SPLINE
SPL {X  -141.803, Y  +311.593, Z    +0.000, E1   +37.608, E3 +232094.448}
SPL {X  -154.548, Y  +344.290, Z    +0.000, E1   +25.264, E3 +232118.932}
SPL {X  -159.249, Y  +370.212, Z    +0.000, E1   +11.801, E3 +232126.964}
SPL {X  -159.987, Y  +383.623, Z    +0.000, E1    +3.169, E3 +232128.717}
SPL {X  -160.000, Y  +388.238, Z    +0.000, E1    -0.420, E3 +232128.928}
SPL {X  -160.000, Y  +392.418, Z    +0.000, E1    -5.131, E3 +232129.169}
SPL {X  -160.000, Y  +399.157, Z    +0.000, E1   -14.351, E3 +232129.985}
SPL {X  -160.000, Y  +411.277, Z    +0.000, E1   -30.487, E3 +232132.763}
SPL {X  -160.000, Y  +452.990, Z    +0.000, E1   -53.470, E3 +232154.127}
SPL {X  -160.000, Y  +539.177, Z    +0.000, E1   -59.280, E3 +232232.454}
SPL {X  -160.000, Y  +554.731, Z    +0.000, E1   -59.281, E3 +232252.098}
SPL {X  -160.000, Y  +572.172, Z    +0.000, E1   -59.312, E3 +232274.061}
SPL {X  -160.000, Y  +589.502, Z    +0.000, E1   -59.284, E3 +232295.999}
SPL {X  -160.000, Y  +604.577, Z    +0.000, E1   -59.272, E3 +232315.058}
SPL {X  -160.000, Y  +620.386, Z    +0.000, E1   -59.294, E3 +232334.986}
SPL {X  -160.000, Y  +636.664, Z    +0.000, E1   -59.282, E3 +232355.575}
SPL {X  -160.000, Y  +654.257, Z    +0.000, E1   -59.312, E3 +232377.754}
SPL {X  -160.000, Y  +671.385, Z    +0.000, E1   -59.278, E3 +232399.443}
SPL {X  -159.497, Y  +687.081, Z    +0.000, E1   -59.218, E3 +232419.770}
SPL {X  -157.563, Y  +702.220, Z    +0.000, E1   -58.916, E3 +232440.931}
SPL {X  -154.922, Y  +714.390, Z    +0.000, E1   -58.446, E3 +232459.125}
SPL {X  -151.559, Y  +725.681, Z    +0.000, E1   -57.922, E3 +232476.756}
SPL {X  -147.777, Y  +735.736, Z    +0.000, E1   -57.226, E3 +232493.250}
SPL {X  -143.698, Y  +744.763, Z    +0.000, E1   -56.526, E3 +232508.527}
SPL {X  -138.992, Y  +753.654, Z    +0.000, E1   -55.630, E3 +232524.104}
SPL {X  -122.847, Y  +776.912, Z    +0.000, E1   -47.251, E3 +232633.787}
ENDSPLINE

SPLINE
SPL {X  -149.319, Y  +731.879, Z    +0.000, E1   -32.249, E3 +232728.173}
SPL {X  -158.304, Y  +697.637, Z    +0.000, E1   -16.440, E3 +232742.824}
SPL {X  -159.863, Y  +681.030, Z    +0.000, E1    -6.312, E3 +232745.766}
SPL {X  -160.000, Y  +673.530, Z    +0.000, E1    -1.059, E3 +232746.273}
SPL {X  -160.000, Y  +670.245, Z    +0.000, E1    +2.042, E3 +232746.386}
SPL {X  -160.000, Y  +663.790, Z    +0.000, E1   +10.467, E3 +232746.911}
SPL {X  -160.000, Y  +655.457, Z    +0.000, E1   +22.866, E3 +232748.273}
SPL {X  -160.000, Y  +644.540, Z    +0.000, E1   +36.054, E3 +232751.304}
SPL {X  -160.000, Y  +601.495, Z    +0.000, E1   +56.174, E3 +232772.233}
SPL {X  -160.000, Y  +515.545, Z    +0.000, E1   +60.629, E3 +232847.627}
SPL {X  -160.000, Y  +503.330, Z    +0.000, E1   +60.630, E3 +232862.233}
SPL {X  -160.000, Y  +487.139, Z    +0.000, E1   +60.676, E3 +232881.501}
SPL {X  -160.000, Y  +466.770, Z    +0.000, E1   +60.698, E3 +232905.797}
SPL {X  -160.000, Y  +454.269, Z    +0.000, E1   +59.898, E3 +232926.048}
ENDSPLINE

SPLINE
SPL {X  -160.000, Y  +458.973, Z    +0.000, E1   +55.880, E3 +232946.966}
ENDSPLINE

SPLINE
SPL {X  -160.000, Y  +435.816, Z    +0.000, E1   +57.237, E3 +232970.642}
SPL {X  -160.000, Y  +411.824, Z    +0.000, E1   +58.675, E3 +232993.135}
SPL {X  -160.000, Y  +390.940, Z    +0.000, E1   +59.356, E3 +233015.163}
SPL {X  -159.620, Y  +374.678, Z    +0.000, E1   +59.299, E3 +233036.047}
SPL {X  -157.749, Y  +358.956, Z    +0.000, E1   +59.037, E3 +233057.745}
SPL {X  -154.809, Y  +345.275, Z    +0.000, E1   +58.527, E3 +233078.068}
SPL {X  -151.181, Y  +333.313, Z    +0.000, E1   +57.939, E3 +233096.777}
SPL {X  -146.730, Y  +321.901, Z    +0.000, E1   +57.169, E3 +233115.522}
SPL {X  -142.568, Y  +313.075, Z    +0.000, E1   +56.366, E3 +233130.644}
SPL {X  -139.172, Y  +306.763, Z    +0.000, E1   +55.717, E3 +233141.699}
SPL {X  -137.037, Y  +303.112, Z    +0.000, E1   +55.261, E3 +233148.245}
SPL {X  -123.439, Y  +283.902, Z    +0.000, E1   +48.158, E3 +233234.596}
ENDSPLINE

SPLINE
SPL {X  -141.803, Y  +311.593, Z    +0.000, E1   +37.608, E3 +233325.216}
SPL {X  -154.548, Y  +344.290, Z    +0.000, E1   +25.264, E3 +233349.699}
SPL {X  -159.249, Y  +370.212, Z    +0.000, E1   +11.801, E3 +233357.731}
SPL {X  -159.987, Y  +383.623, Z    +0.000, E1    +3.169, E3 +233359.484}
SPL {X  -160.000, Y  +388.238, Z    +0.000, E1    -0.420, E3 +233359.696}
SPL {X  -160.000, Y  +392.418, Z    +0.000, E1    -5.131, E3 +233359.936}
SPL {X  -160.000, Y  +399.157, Z    +0.000, E1   -14.351, E3 +233360.752}
SPL {X  -160.000, Y  +411.277, Z    +0.000, E1   -30.487, E3 +233363.530}
SPL {X  -160.000, Y  +452.990, Z    +0.000, E1   -53.470, E3 +233384.894}
SPL {X  -160.000, Y  +539.177, Z    +0.000, E1   -59.280, E3 +233463.221}
SPL {X  -160.000, Y  +554.731, Z    +0.000, E1   -59.281, E3 +233482.865}
SPL {X  -160.000, Y  +572.172, Z    +0.000, E1   -59.312, E3 +233504.828}
SPL {X  -160.000, Y  +589.502, Z    +0.000, E1   -59.284, E3 +233526.766}
SPL {X  -160.000, Y  +604.577, Z    +0.000, E1   -59.272, E3 +233545.826}
SPL {X  -160.000, Y  +620.386, Z    +0.000, E1   -59.294, E3 +233565.753}
SPL {X  -160.000, Y  +636.664, Z    +0.000, E1   -59.282, E3 +233586.343}
SPL {X  -160.000, Y  +654.257, Z    +0.000, E1   -59.312, E3 +233608.521}
SPL {X  -160.000, Y  +671.385, Z    +0.000, E1   -59.278, E3 +233630.210}
SPL {X  -159.497, Y  +687.081, Z    +0.000, E1   -59.218, E3 +233650.537}
SPL {X  -157.563, Y  +702.220, Z    +0.000, E1   -58.916, E3 +233671.699}
SPL {X  -154.922, Y  +714.390, Z    +0.000, E1   -58.446, E3 +233689.892}
SPL {X  -151.559, Y  +725.681, Z    +0.000, E1   -57.922, E3 +233707.523}
SPL {X  -147.777, Y  +735.736, Z    +0.000, E1   -57.226, E3 +233724.017}
SPL {X  -143.698, Y  +744.763, Z    +0.000, E1   -56.526, E3 +233739.294}
SPL {X  -138.992, Y  +753.654, Z    +0.000, E1   -55.630, E3 +233754.871}
SPL {X  -122.847, Y  +776.912, Z    +0.000, E1   -47.251, E3 +233864.554}
ENDSPLINE

SPLINE
SPL {X  -149.319, Y  +731.879, Z    +0.000, E1   -32.249, E3 +233958.941}
SPL {X  -158.304, Y  +697.637, Z    +0.000, E1   -16.440, E3 +233973.591}
SPL {X  -159.863, Y  +681.030, Z    +0.000, E1    -6.312, E3 +233976.533}
SPL {X  -160.000, Y  +673.530, Z    +0.000, E1    -1.059, E3 +233977.040}
SPL {X  -160.000, Y  +670.245, Z    +0.000, E1    +2.042, E3 +233977.153}
SPL {X  -160.000, Y  +663.790, Z    +0.000, E1   +10.467, E3 +233977.678}
SPL {X  -160.000, Y  +655.457, Z    +0.000, E1   +22.866, E3 +233979.040}
SPL {X  -160.000, Y  +644.540, Z    +0.000, E1   +36.054, E3 +233982.071}
SPL {X  -160.000, Y  +601.495, Z    +0.000, E1   +56.174, E3 +234003.000}
SPL {X  -160.000, Y  +515.545, Z    +0.000, E1   +60.629, E3 +234078.394}
SPL {X  -160.000, Y  +503.330, Z    +0.000, E1   +60.630, E3 +234093.000}
SPL {X  -160.000, Y  +487.139, Z    +0.000, E1   +60.676, E3 +234112.268}
SPL {X  -160.000, Y  +466.770, Z    +0.000, E1   +60.698, E3 +234136.564}
SPL {X  -160.000, Y  +454.269, Z    +0.000, E1   +59.898, E3 +234156.815}
ENDSPLINE

SPLINE
SPL {X  -160.000, Y  +458.973, Z    +0.000, E1   +55.880, E3 +234177.733}
ENDSPLINE

SPLINE
SPL {X  -160.000, Y  +435.816, Z    +0.000, E1   +57.237, E3 +234201.409}
SPL {X  -160.000, Y  +411.824, Z    +0.000, E1   +58.675, E3 +234223.903}
SPL {X  -160.000, Y  +390.940, Z    +0.000, E1   +59.356, E3 +234245.930}
SPL {X  -159.620, Y  +374.678, Z    +0.000, E1   +59.299, E3 +234266.814}
SPL {X  -157.749, Y  +358.956, Z    +0.000, E1   +59.037, E3 +234288.512}
SPL {X  -154.809, Y  +345.275, Z    +0.000, E1   +58.527, E3 +234308.835}
SPL {X  -151.181, Y  +333.313, Z    +0.000, E1   +57.939, E3 +234327.544}
SPL {X  -146.730, Y  +321.901, Z    +0.000, E1   +57.169, E3 +234346.289}
SPL {X  -142.568, Y  +313.075, Z    +0.000, E1   +56.366, E3 +234361.411}
SPL {X  -139.172, Y  +306.763, Z    +0.000, E1   +55.717, E3 +234372.466}
SPL {X  -137.037, Y  +303.112, Z    +0.000, E1   +55.261, E3 +234379.012}
SPL {X  -123.439, Y  +283.902, Z    +0.000, E1   +48.158, E3 +234465.364}
ENDSPLINE

SPLINE
SPL {X  -141.803, Y  +311.593, Z    +0.000, E1   +37.608, E3 +234555.983}
SPL {X  -154.548, Y  +344.290, Z    +0.000, E1   +25.264, E3 +234580.466}
SPL {X  -159.249, Y  +370.212, Z    +0.000, E1   +11.801, E3 +234588.498}
SPL {X  -159.987, Y  +383.623, Z    +0.000, E1    +3.169, E3 +234590.251}
SPL {X  -160.000, Y  +388.238, Z    +0.000, E1    -0.420, E3 +234590.463}
SPL {X  -160.000, Y  +392.418, Z    +0.000, E1    -5.131, E3 +234590.703}
SPL {X  -160.000, Y  +399.157, Z    +0.000, E1   -14.351, E3 +234591.520}
SPL {X  -160.000, Y  +411.277, Z    +0.000, E1   -30.487, E3 +234594.298}
SPL {X  -160.000, Y  +452.990, Z    +0.000, E1   -53.470, E3 +234615.662}
SPL {X  -160.000, Y  +539.177, Z    +0.000, E1   -59.280, E3 +234693.988}
SPL {X  -160.000, Y  +554.731, Z    +0.000, E1   -59.281, E3 +234713.633}
SPL {X  -160.000, Y  +572.172, Z    +0.000, E1   -59.312, E3 +234735.595}
SPL {X  -160.000, Y  +589.502, Z    +0.000, E1   -59.284, E3 +234757.534}
SPL {X  -160.000, Y  +604.577, Z    +0.000, E1   -59.272, E3 +234776.593}
SPL {X  -160.000, Y  +620.386, Z    +0.000, E1   -59.294, E3 +234796.520}
SPL {X  -160.000, Y  +636.664, Z    +0.000, E1   -59.282, E3 +234817.110}
SPL {X  -160.000, Y  +654.257, Z    +0.000, E1   -59.312, E3 +234839.288}
SPL {X  -160.000, Y  +671.385, Z    +0.000, E1   -59.278, E3 +234860.977}
SPL {X  -159.497, Y  +687.081, Z    +0.000, E1   -59.218, E3 +234881.304}
SPL {X  -157.563, Y  +702.220, Z    +0.000, E1   -58.916, E3 +234902.466}
SPL {X  -154.922, Y  +714.390, Z    +0.000, E1   -58.446, E3 +234920.659}
SPL {X  -151.559, Y  +725.681, Z    +0.000, E1   -57.922, E3 +234938.290}
SPL {X  -147.777, Y  +735.736, Z    +0.000, E1   -57.226, E3 +234954.785}
SPL {X  -143.698, Y  +744.763, Z    +0.000, E1   -56.526, E3 +234970.061}
SPL {X  -138.992, Y  +753.654, Z    +0.000, E1   -55.630, E3 +234985.638}
SPL {X  -122.847, Y  +776.912, Z    +0.000, E1   -47.251, E3 +235095.321}
ENDSPLINE

SPLINE
SPL {X  -149.319, Y  +731.879, Z    +0.000, E1   -32.249, E3 +235189.708}
SPL {X  -158.304, Y  +697.637, Z    +0.000, E1   -16.440, E3 +235204.358}
SPL {X  -159.863, Y  +681.030, Z    +0.000, E1    -6.312, E3 +235207.301}
SPL {X  -160.000, Y  +673.530, Z    +0.000, E1    -1.059, E3 +235207.807}
SPL {X  -160.000, Y  +670.245, Z    +0.000, E1    +2.042, E3 +235207.921}
SPL {X  -160.000, Y  +663.790, Z    +0.000, E1   +10.467, E3 +235208.445}
SPL {X  -160.000, Y  +655.457, Z    +0.000, E1   +22.866, E3 +235209.807}
SPL {X  -160.000, Y  +644.540, Z    +0.000, E1   +36.054, E3 +235212.838}
SPL {X  -160.000, Y  +601.495, Z    +0.000, E1   +56.174, E3 +235233.768}
SPL {X  -160.000, Y  +515.545, Z    +0.000, E1   +60.629, E3 +235309.162}
SPL {X  -160.000, Y  +503.330, Z    +0.000, E1   +60.630, E3 +235323.767}
SPL {X  -160.000, Y  +487.139, Z    +0.000, E1   +60.676, E3 +235343.036}
SPL {X  -160.000, Y  +466.770, Z    +0.000, E1   +60.698, E3 +235367.331}
SPL {X  -160.000, Y  +454.269, Z    +0.000, E1   +59.898, E3 +235387.582}
ENDSPLINE

SPLINE
SPL {X  -160.000, Y  +458.973, Z    +0.000, E1   +55.880, E3 +235408.501}
ENDSPLINE

SPLINE
SPL {X  -160.000, Y  +435.816, Z    +0.000, E1   +57.237, E3 +235432.176}
SPL {X  -160.000, Y  +411.824, Z    +0.000, E1   +58.675, E3 +235454.670}
SPL {X  -160.000, Y  +390.940, Z    +0.000, E1   +59.356, E3 +235476.698}
SPL {X  -159.620, Y  +374.678, Z    +0.000, E1   +59.299, E3 +235497.581}
SPL {X  -157.749, Y  +358.956, Z    +0.000, E1   +59.037, E3 +235519.279}
SPL {X  -154.809, Y  +345.275, Z    +0.000, E1   +58.527, E3 +235539.603}
SPL {X  -151.181, Y  +333.313, Z    +0.000, E1   +57.939, E3 +235558.311}
SPL {X  -146.730, Y  +321.901, Z    +0.000, E1   +57.169, E3 +235577.057}
SPL {X  -142.568, Y  +313.075, Z    +0.000, E1   +56.366, E3 +235592.178}
SPL {X  -138.721, Y  +305.972, Z    +0.000, E1   +55.652, E3 +235604.606}
SPL {X  -123.439, Y  +283.902, Z    +0.000, E1   +48.158, E3 +235696.131}
ENDSPLINE

SPLINE
SPL {X  -141.803, Y  +311.593, Z    +0.000, E1   +37.608, E3 +235786.750}
SPL {X  -154.548, Y  +344.290, Z    +0.000, E1   +25.264, E3 +235811.233}
SPL {X  -159.249, Y  +370.212, Z    +0.000, E1   +11.801, E3 +235819.266}
SPL {X  -159.987, Y  +383.623, Z    +0.000, E1    +3.169, E3 +235821.019}
SPL {X  -160.000, Y  +388.238, Z    +0.000, E1    -0.420, E3 +235821.230}
SPL {X  -160.000, Y  +392.418, Z    +0.000, E1    -5.131, E3 +235821.470}
SPL {X  -160.000, Y  +399.157, Z    +0.000, E1   -14.351, E3 +235822.287}
SPL {X  -160.000, Y  +411.277, Z    +0.000, E1   -30.487, E3 +235825.065}
SPL {X  -160.000, Y  +452.990, Z    +0.000, E1   -53.470, E3 +235846.429}
SPL {X  -160.000, Y  +539.177, Z    +0.000, E1   -59.280, E3 +235924.755}
SPL {X  -160.000, Y  +554.731, Z    +0.000, E1   -59.281, E3 +235944.400}
SPL {X  -160.000, Y  +572.172, Z    +0.000, E1   -59.312, E3 +235966.363}
SPL {X  -160.000, Y  +589.502, Z    +0.000, E1   -59.284, E3 +235988.301}
SPL {X  -160.000, Y  +604.577, Z    +0.000, E1   -59.272, E3 +236007.360}
SPL {X  -160.000, Y  +620.386, Z    +0.000, E1   -59.294, E3 +236027.287}
SPL {X  -160.000, Y  +636.664, Z    +0.000, E1   -59.282, E3 +236047.877}
SPL {X  -160.000, Y  +654.257, Z    +0.000, E1   -59.312, E3 +236070.055}
SPL {X  -160.000, Y  +671.385, Z    +0.000, E1   -59.278, E3 +236091.744}
SPL {X  -159.497, Y  +687.081, Z    +0.000, E1   -59.218, E3 +236112.072}
SPL {X  -157.563, Y  +702.220, Z    +0.000, E1   -58.916, E3 +236133.233}
SPL {X  -154.922, Y  +714.390, Z    +0.000, E1   -58.446, E3 +236151.427}
SPL {X  -151.559, Y  +725.681, Z    +0.000, E1   -57.922, E3 +236169.057}
SPL {X  -147.777, Y  +735.736, Z    +0.000, E1   -57.226, E3 +236185.552}
SPL {X  -143.698, Y  +744.763, Z    +0.000, E1   -56.526, E3 +236200.828}
SPL {X  -138.992, Y  +753.654, Z    +0.000, E1   -55.630, E3 +236216.406}
SPL {X  -122.847, Y  +776.912, Z    +0.000, E1   -47.251, E3 +236326.088}
ENDSPLINE

SPLINE
SPL {X  -149.319, Y  +731.879, Z    +0.000, E1   -32.249, E3 +236420.475}
SPL {X  -158.304, Y  +697.637, Z    +0.000, E1   -16.440, E3 +236435.126}
SPL {X  -159.863, Y  +681.030, Z    +0.000, E1    -6.312, E3 +236438.068}
SPL {X  -160.000, Y  +673.530, Z    +0.000, E1    -1.059, E3 +236438.575}
SPL {X  -160.000, Y  +670.245, Z    +0.000, E1    +2.042, E3 +236438.688}
SPL {X  -160.000, Y  +663.790, Z    +0.000, E1   +10.467, E3 +236439.212}
SPL {X  -160.000, Y  +655.457, Z    +0.000, E1   +22.866, E3 +236440.575}
SPL {X  -160.000, Y  +644.540, Z    +0.000, E1   +36.054, E3 +236443.606}
SPL {X  -160.000, Y  +601.495, Z    +0.000, E1   +56.174, E3 +236464.535}
SPL {X  -160.000, Y  +515.545, Z    +0.000, E1   +60.629, E3 +236539.929}
SPL {X  -160.000, Y  +503.330, Z    +0.000, E1   +60.630, E3 +236554.535}
SPL {X  -160.000, Y  +487.139, Z    +0.000, E1   +60.676, E3 +236573.803}
SPL {X  -160.000, Y  +466.770, Z    +0.000, E1   +60.698, E3 +236598.098}
SPL {X  -160.000, Y  +454.269, Z    +0.000, E1   +59.898, E3 +236618.349}
ENDSPLINE

SPLINE
SPL {X  -160.000, Y  +458.973, Z    +0.000, E1   +55.880, E3 +236639.268}
ENDSPLINE

SPLINE
SPL {X  -160.000, Y  +435.816, Z    +0.000, E1   +57.237, E3 +236662.943}
SPL {X  -160.000, Y  +411.824, Z    +0.000, E1   +58.675, E3 +236685.437}
SPL {X  -160.000, Y  +390.940, Z    +0.000, E1   +59.356, E3 +236707.465}
SPL {X  -159.620, Y  +374.678, Z    +0.000, E1   +59.299, E3 +236728.349}
SPL {X  -157.749, Y  +358.956, Z    +0.000, E1   +59.037, E3 +236750.047}
SPL {X  -154.809, Y  +345.275, Z    +0.000, E1   +58.527, E3 +236770.370}
SPL {X  -151.181, Y  +333.313, Z    +0.000, E1   +57.939, E3 +236789.078}
SPL {X  -146.730, Y  +321.901, Z    +0.000, E1   +57.169, E3 +236807.824}
SPL {X  -142.568, Y  +313.075, Z    +0.000, E1   +56.366, E3 +236822.946}
SPL {X  -138.721, Y  +305.972, Z    +0.000, E1   +55.652, E3 +236835.374}
SPL {X  -123.439, Y  +283.902, Z    +0.000, E1   +48.158, E3 +236926.898}
ENDSPLINE

SPLINE
SPL {X  -141.803, Y  +311.593, Z    +0.000, E1   +37.608, E3 +237017.517}
SPL {X  -154.548, Y  +344.290, Z    +0.000, E1   +25.264, E3 +237042.001}
SPL {X  -159.249, Y  +370.212, Z    +0.000, E1   +11.801, E3 +237050.033}
SPL {X  -159.987, Y  +383.623, Z    +0.000, E1    +3.169, E3 +237051.786}
SPL {X  -160.000, Y  +388.238, Z    +0.000, E1    -0.420, E3 +237051.997}
SPL {X  -160.000, Y  +392.418, Z    +0.000, E1    -5.131, E3 +237052.238}
SPL {X  -160.000, Y  +399.157, Z    +0.000, E1   -14.351, E3 +237053.054}
SPL {X  -160.000, Y  +411.277, Z    +0.000, E1   -30.487, E3 +237055.832}
SPL {X  -160.000, Y  +452.990, Z    +0.000, E1   -53.470, E3 +237077.196}
SPL {X  -160.000, Y  +539.177, Z    +0.000, E1   -59.280, E3 +237155.523}
SPL {X  -160.000, Y  +554.731, Z    +0.000, E1   -59.281, E3 +237175.167}
SPL {X  -160.000, Y  +572.172, Z    +0.000, E1   -59.312, E3 +237197.130}
SPL {X  -160.000, Y  +589.502, Z    +0.000, E1   -59.284, E3 +237219.068}
SPL {X  -160.000, Y  +604.577, Z    +0.000, E1   -59.272, E3 +237238.127}
SPL {X  -160.000, Y  +620.386, Z    +0.000, E1   -59.294, E3 +237258.055}
SPL {X  -160.000, Y  +636.664, Z    +0.000, E1   -59.282, E3 +237278.644}
SPL {X  -160.000, Y  +654.257, Z    +0.000, E1   -59.312, E3 +237300.823}
SPL {X  -160.000, Y  +671.385, Z    +0.000, E1   -59.278, E3 +237322.512}
SPL {X  -159.497, Y  +687.081, Z    +0.000, E1   -59.218, E3 +237342.839}
SPL {X  -157.563, Y  +702.220, Z    +0.000, E1   -58.916, E3 +237364.000}
SPL {X  -154.922, Y  +714.390, Z    +0.000, E1   -58.446, E3 +237382.194}
SPL {X  -151.559, Y  +725.681, Z    +0.000, E1   -57.922, E3 +237399.825}
SPL {X  -147.777, Y  +735.736, Z    +0.000, E1   -57.226, E3 +237416.319}
SPL {X  -143.698, Y  +744.763, Z    +0.000, E1   -56.526, E3 +237431.596}
SPL {X  -138.992, Y  +753.654, Z    +0.000, E1   -55.630, E3 +237447.173}
SPL {X  -122.847, Y  +776.912, Z    +0.000, E1   -47.251, E3 +237556.856}
ENDSPLINE

SPLINE
SPL {X  -149.319, Y  +731.879, Z    +0.000, E1   -32.249, E3 +237651.242}
SPL {X  -158.304, Y  +697.637, Z    +0.000, E1   -16.440, E3 +237665.893}
SPL {X  -159.863, Y  +681.030, Z    +0.000, E1    -6.312, E3 +237668.835}
SPL {X  -160.000, Y  +673.530, Z    +0.000, E1    -1.059, E3 +237669.342}
SPL {X  -160.000, Y  +670.245, Z    +0.000, E1    +2.042, E3 +237669.455}
SPL {X  -160.000, Y  +663.790, Z    +0.000, E1   +10.467, E3 +237669.980}
SPL {X  -160.000, Y  +655.457, Z    +0.000, E1   +22.866, E3 +237671.342}
SPL {X  -160.000, Y  +644.540, Z    +0.000, E1   +36.054, E3 +237674.373}
SPL {X  -160.000, Y  +601.495, Z    +0.000, E1   +56.174, E3 +237695.302}
SPL {X  -160.000, Y  +515.545, Z    +0.000, E1   +60.629, E3 +237770.696}
SPL {X  -160.000, Y  +503.330, Z    +0.000, E1   +60.630, E3 +237785.302}
SPL {X  -160.000, Y  +487.139, Z    +0.000, E1   +60.676, E3 +237804.570}
SPL {X  -160.000, Y  +466.770, Z    +0.000, E1   +60.698, E3 +237828.866}
SPL {X  -160.000, Y  +454.269, Z    +0.000, E1   +59.898, E3 +237849.117}
ENDSPLINE

SPLINE
SPL {X  -160.000, Y  +458.973, Z    +0.000, E1   +55.880, E3 +237870.035}
ENDSPLINE

SPLINE
SPL {X  -160.000, Y  +435.816, Z    +0.000, E1   +57.237, E3 +237893.711}
SPL {X  -160.000, Y  +411.824, Z    +0.000, E1   +58.675, E3 +237916.204}
SPL {X  -160.000, Y  +390.940, Z    +0.000, E1   +59.356, E3 +237938.232}
SPL {X  -159.620, Y  +374.678, Z    +0.000, E1   +59.299, E3 +237959.116}
SPL {X  -157.749, Y  +358.956, Z    +0.000, E1   +59.037, E3 +237980.814}
SPL {X  -154.809, Y  +345.275, Z    +0.000, E1   +58.527, E3 +238001.137}
SPL {X  -151.181, Y  +333.313, Z    +0.000, E1   +57.939, E3 +238019.846}
SPL {X  -146.730, Y  +321.901, Z    +0.000, E1   +57.169, E3 +238038.591}
SPL {X  -142.568, Y  +313.075, Z    +0.000, E1   +56.366, E3 +238053.713}
SPL {X  -139.172, Y  +306.763, Z    +0.000, E1   +55.717, E3 +238064.768}
SPL {X  -137.037, Y  +303.112, Z    +0.000, E1   +55.261, E3 +238071.314}
SPL {X  -123.439, Y  +283.902, Z    +0.000, E1   +48.158, E3 +238157.665}
ENDSPLINE

SPLINE
SPL {X  -141.803, Y  +311.593, Z    +0.000, E1   +37.608, E3 +238248.285}
SPL {X  -154.548, Y  +344.290, Z    +0.000, E1   +25.264, E3 +238272.768}
SPL {X  -159.249, Y  +370.212, Z    +0.000, E1   +11.801, E3 +238280.800}
SPL {X  -159.987, Y  +383.623, Z    +0.000, E1    +3.169, E3 +238282.553}
SPL {X  -160.000, Y  +388.238, Z    +0.000, E1    -0.420, E3 +238282.765}
SPL {X  -160.000, Y  +392.418, Z    +0.000, E1    -5.131, E3 +238283.005}
SPL {X  -160.000, Y  +399.157, Z    +0.000, E1   -14.351, E3 +238283.821}
SPL {X  -160.000, Y  +411.277, Z    +0.000, E1   -30.487, E3 +238286.599}
SPL {X  -160.000, Y  +452.990, Z    +0.000, E1   -53.470, E3 +238307.963}
SPL {X  -160.000, Y  +539.177, Z    +0.000, E1   -59.280, E3 +238386.290}
SPL {X  -160.000, Y  +554.731, Z    +0.000, E1   -59.281, E3 +238405.934}
SPL {X  -160.000, Y  +572.172, Z    +0.000, E1   -59.312, E3 +238427.897}
SPL {X  -160.000, Y  +589.502, Z    +0.000, E1   -59.284, E3 +238449.835}
SPL {X  -160.000, Y  +604.577, Z    +0.000, E1   -59.272, E3 +238468.895}
SPL {X  -160.000, Y  +620.386, Z    +0.000, E1   -59.294, E3 +238488.822}
SPL {X  -160.000, Y  +636.664, Z    +0.000, E1   -59.282, E3 +238509.412}
SPL {X  -160.000, Y  +654.257, Z    +0.000, E1   -59.312, E3 +238531.590}
SPL {X  -160.000, Y  +671.385, Z    +0.000, E1   -59.278, E3 +238553.279}
SPL {X  -159.497, Y  +687.081, Z    +0.000, E1   -59.218, E3 +238573.606}
SPL {X  -157.563, Y  +702.220, Z    +0.000, E1   -58.916, E3 +238594.768}
SPL {X  -154.922, Y  +714.390, Z    +0.000, E1   -58.446, E3 +238612.961}
SPL {X  -151.559, Y  +725.681, Z    +0.000, E1   -57.922, E3 +238630.592}
SPL {X  -147.777, Y  +735.736, Z    +0.000, E1   -57.226, E3 +238647.087}
SPL {X  -143.698, Y  +744.763, Z    +0.000, E1   -56.526, E3 +238662.363}
SPL {X  -138.992, Y  +753.654, Z    +0.000, E1   -55.630, E3 +238677.940}
SPL {X  -122.847, Y  +776.912, Z    +0.000, E1   -47.251, E3 +238787.623}
ENDSPLINE

SPLINE
SPL {X  -149.319, Y  +731.879, Z    +0.000, E1   -32.249, E3 +238882.010}
SPL {X  -158.304, Y  +697.637, Z    +0.000, E1   -16.440, E3 +238896.660}
SPL {X  -159.863, Y  +681.030, Z    +0.000, E1    -6.312, E3 +238899.602}
SPL {X  -160.000, Y  +673.530, Z    +0.000, E1    -1.059, E3 +238900.109}
SPL {X  -160.000, Y  +670.245, Z    +0.000, E1    +2.042, E3 +238900.222}
SPL {X  -160.000, Y  +663.790, Z    +0.000, E1   +10.467, E3 +238900.747}
SPL {X  -160.000, Y  +655.457, Z    +0.000, E1   +22.866, E3 +238902.109}
SPL {X  -160.000, Y  +644.540, Z    +0.000, E1   +36.054, E3 +238905.140}
SPL {X  -160.000, Y  +601.495, Z    +0.000, E1   +56.174, E3 +238926.069}
SPL {X  -160.000, Y  +515.545, Z    +0.000, E1   +60.629, E3 +239001.463}
SPL {X  -160.000, Y  +503.330, Z    +0.000, E1   +60.630, E3 +239016.069}
SPL {X  -160.000, Y  +487.139, Z    +0.000, E1   +60.676, E3 +239035.337}
SPL {X  -160.000, Y  +466.770, Z    +0.000, E1   +60.698, E3 +239059.633}
SPL {X  -160.000, Y  +454.269, Z    +0.000, E1   +59.898, E3 +239079.884}
ENDSPLINE

SPLINE
SPL {X  -160.000, Y  +458.973, Z    +0.000, E1   +55.880, E3 +239100.802}
ENDSPLINE

SPLINE
SPL {X  -160.000, Y  +435.816, Z    +0.000, E1   +57.237, E3 +239124.478}
SPL {X  -160.000, Y  +411.824, Z    +0.000, E1   +58.675, E3 +239146.972}
SPL {X  -160.000, Y  +390.940, Z    +0.000, E1   +59.356, E3 +239168.999}
SPL {X  -159.620, Y  +374.678, Z    +0.000, E1   +59.299, E3 +239189.883}
SPL {X  -157.749, Y  +358.956, Z    +0.000, E1   +59.037, E3 +239211.581}
SPL {X  -154.809, Y  +345.275, Z    +0.000, E1   +58.527, E3 +239231.904}
SPL {X  -151.181, Y  +333.313, Z    +0.000, E1   +57.939, E3 +239250.613}
SPL {X  -146.730, Y  +321.901, Z    +0.000, E1   +57.169, E3 +239269.358}
SPL {X  -142.568, Y  +313.075, Z    +0.000, E1   +56.366, E3 +239284.480}
SPL {X  -139.172, Y  +306.763, Z    +0.000, E1   +55.717, E3 +239295.535}
SPL {X  -137.037, Y  +303.112, Z    +0.000, E1   +55.261, E3 +239302.081}
SPL {X  -123.439, Y  +283.902, Z    +0.000, E1   +48.158, E3 +239388.433}
ENDSPLINE

SPLINE
SPL {X  -141.803, Y  +311.593, Z    +0.000, E1   +37.608, E3 +239479.052}
SPL {X  -154.548, Y  +344.290, Z    +0.000, E1   +25.264, E3 +239503.535}
SPL {X  -159.249, Y  +370.212, Z    +0.000, E1   +11.801, E3 +239511.567}
SPL {X  -159.987, Y  +383.623, Z    +0.000, E1    +3.169, E3 +239513.320}
SPL {X  -160.000, Y  +388.238, Z    +0.000, E1    -0.420, E3 +239513.532}
SPL {X  -160.000, Y  +392.418, Z    +0.000, E1    -5.131, E3 +239513.772}
SPL {X  -160.000, Y  +399.157, Z    +0.000, E1   -14.351, E3 +239514.589}
SPL {X  -160.000, Y  +411.277, Z    +0.000, E1   -30.487, E3 +239517.367}
SPL {X  -160.000, Y  +452.990, Z    +0.000, E1   -53.470, E3 +239538.731}
SPL {X  -160.000, Y  +539.177, Z    +0.000, E1   -59.280, E3 +239617.057}
SPL {X  -160.000, Y  +554.731, Z    +0.000, E1   -59.281, E3 +239636.702}
SPL {X  -160.000, Y  +572.172, Z    +0.000, E1   -59.312, E3 +239658.664}
SPL {X  -160.000, Y  +589.502, Z    +0.000, E1   -59.284, E3 +239680.603}
SPL {X  -160.000, Y  +604.577, Z    +0.000, E1   -59.272, E3 +239699.662}
SPL {X  -160.000, Y  +620.386, Z    +0.000, E1   -59.294, E3 +239719.589}
SPL {X  -160.000, Y  +636.664, Z    +0.000, E1   -59.282, E3 +239740.179}
SPL {X  -160.000, Y  +654.257, Z    +0.000, E1   -59.312, E3 +239762.357}
SPL {X  -160.000, Y  +671.385, Z    +0.000, E1   -59.278, E3 +239784.046}
SPL {X  -159.497, Y  +687.081, Z    +0.000, E1   -59.218, E3 +239804.373}
SPL {X  -157.563, Y  +702.220, Z    +0.000, E1   -58.916, E3 +239825.535}
SPL {X  -154.922, Y  +714.390, Z    +0.000, E1   -58.446, E3 +239843.729}
SPL {X  -151.559, Y  +725.681, Z    +0.000, E1   -57.922, E3 +239861.359}
SPL {X  -147.777, Y  +735.736, Z    +0.000, E1   -57.226, E3 +239877.854}
SPL {X  -143.698, Y  +744.763, Z    +0.000, E1   -56.526, E3 +239893.130}
SPL {X  -138.992, Y  +753.654, Z    +0.000, E1   -55.630, E3 +239908.707}
SPL {X  -122.847, Y  +776.912, Z    +0.000, E1   -47.251, E3 +240018.390}
ENDSPLINE

SPLINE
SPL {X  -149.319, Y  +731.879, Z    +0.000, E1   -32.249, E3 +240112.777}
SPL {X  -158.304, Y  +697.637, Z    +0.000, E1   -16.440, E3 +240127.427}
SPL {X  -159.863, Y  +681.030, Z    +0.000, E1    -6.312, E3 +240130.370}
SPL {X  -160.000, Y  +673.530, Z    +0.000, E1    -1.059, E3 +240130.876}
SPL {X  -160.000, Y  +670.245, Z    +0.000, E1    +2.042, E3 +240130.990}
SPL {X  -160.000, Y  +663.790, Z    +0.000, E1   +10.467, E3 +240131.514}
SPL {X  -160.000, Y  +655.457, Z    +0.000, E1   +22.866, E3 +240132.876}
SPL {X  -160.000, Y  +644.540, Z    +0.000, E1   +36.054, E3 +240135.907}
SPL {X  -160.000, Y  +601.495, Z    +0.000, E1   +56.174, E3 +240156.837}
SPL {X  -160.000, Y  +515.545, Z    +0.000, E1   +60.629, E3 +240232.231}
SPL {X  -160.000, Y  +503.330, Z    +0.000, E1   +60.630, E3 +240246.836}
SPL {X  -160.000, Y  +487.139, Z    +0.000, E1   +60.676, E3 +240266.105}
SPL {X  -160.000, Y  +466.770, Z    +0.000, E1   +60.698, E3 +240290.400}
SPL {X  -160.000, Y  +454.269, Z    +0.000, E1   +59.898, E3 +240310.651}
ENDSPLINE

SPLINE
SPL {X  -160.000, Y  +458.973, Z    +0.000, E1   +55.880, E3 +240331.570}
ENDSPLINE

SPLINE
SPL {X  -160.000, Y  +435.816, Z    +0.000, E1   +57.237, E3 +240355.245}
SPL {X  -160.000, Y  +411.824, Z    +0.000, E1   +58.675, E3 +240377.739}
SPL {X  -160.000, Y  +390.940, Z    +0.000, E1   +59.356, E3 +240399.767}
SPL {X  -159.620, Y  +374.678, Z    +0.000, E1   +59.299, E3 +240420.650}
SPL {X  -157.749, Y  +358.956, Z    +0.000, E1   +59.037, E3 +240442.348}
SPL {X  -154.809, Y  +345.275, Z    +0.000, E1   +58.527, E3 +240462.672}
SPL {X  -151.181, Y  +333.313, Z    +0.000, E1   +57.939, E3 +240481.380}
SPL {X  -146.730, Y  +321.901, Z    +0.000, E1   +57.169, E3 +240500.126}
SPL {X  -142.568, Y  +313.075, Z    +0.000, E1   +56.366, E3 +240515.247}
SPL {X  -139.172, Y  +306.763, Z    +0.000, E1   +55.717, E3 +240526.302}
SPL {X  -137.037, Y  +303.112, Z    +0.000, E1   +55.261, E3 +240532.849}
SPL {X  -123.439, Y  +283.902, Z    +0.000, E1   +48.158, E3 +240619.200}
ENDSPLINE

SPLINE
SPL {X  -141.803, Y  +311.593, Z    +0.000, E1   +37.608, E3 +240709.819}
SPL {X  -154.548, Y  +344.290, Z    +0.000, E1   +25.264, E3 +240734.302}
SPL {X  -159.249, Y  +370.212, Z    +0.000, E1   +11.801, E3 +240742.335}
SPL {X  -159.987, Y  +383.623, Z    +0.000, E1    +3.169, E3 +240744.088}
SPL {X  -160.000, Y  +388.238, Z    +0.000, E1    -0.420, E3 +240744.299}
SPL {X  -160.000, Y  +392.418, Z    +0.000, E1    -5.131, E3 +240744.539}
SPL {X  -160.000, Y  +399.157, Z    +0.000, E1   -14.351, E3 +240745.356}
SPL {X  -160.000, Y  +411.277, Z    +0.000, E1   -30.487, E3 +240748.134}
SPL {X  -160.000, Y  +452.990, Z    +0.000, E1   -53.470, E3 +240769.498}
SPL {X  -160.000, Y  +539.177, Z    +0.000, E1   -59.280, E3 +240847.825}
SPL {X  -160.000, Y  +554.731, Z    +0.000, E1   -59.281, E3 +240867.469}
SPL {X  -160.000, Y  +572.172, Z    +0.000, E1   -59.312, E3 +240889.432}
SPL {X  -160.000, Y  +589.502, Z    +0.000, E1   -59.284, E3 +240911.370}
SPL {X  -160.000, Y  +604.577, Z    +0.000, E1   -59.272, E3 +240930.429}
SPL {X  -160.000, Y  +620.386, Z    +0.000, E1   -59.294, E3 +240950.356}
SPL {X  -160.000, Y  +636.664, Z    +0.000, E1   -59.282, E3 +240970.946}
SPL {X  -160.000, Y  +654.257, Z    +0.000, E1   -59.312, E3 +240993.124}
SPL {X  -160.000, Y  +671.385, Z    +0.000, E1   -59.278, E3 +241014.813}
SPL {X  -159.497, Y  +687.081, Z    +0.000, E1   -59.218, E3 +241035.141}
SPL {X  -157.563, Y  +702.220, Z    +0.000, E1   -58.916, E3 +241056.302}
SPL {X  -154.922, Y  +714.390, Z    +0.000, E1   -58.446, E3 +241074.496}
SPL {X  -151.559, Y  +725.681, Z    +0.000, E1   -57.922, E3 +241092.126}
SPL {X  -147.777, Y  +735.736, Z    +0.000, E1   -57.226, E3 +241108.621}
SPL {X  -143.698, Y  +744.763, Z    +0.000, E1   -56.526, E3 +241123.897}
SPL {X  -138.992, Y  +753.654, Z    +0.000, E1   -55.630, E3 +241139.475}
SPL {X  -122.847, Y  +776.912, Z    +0.000, E1   -47.251, E3 +241249.157}
ENDSPLINE

SPLINE
SPL {X  -149.319, Y  +731.879, Z    +0.000, E1   -32.249, E3 +241343.544}
SPL {X  -158.304, Y  +697.637, Z    +0.000, E1   -16.440, E3 +241358.195}
SPL {X  -159.863, Y  +681.030, Z    +0.000, E1    -6.312, E3 +241361.137}
SPL {X  -160.000, Y  +673.530, Z    +0.000, E1    -1.059, E3 +241361.644}
SPL {X  -160.000, Y  +670.245, Z    +0.000, E1    +2.042, E3 +241361.757}
SPL {X  -160.000, Y  +663.790, Z    +0.000, E1   +10.467, E3 +241362.281}
SPL {X  -160.000, Y  +655.457, Z    +0.000, E1   +22.866, E3 +241363.644}
SPL {X  -160.000, Y  +644.540, Z    +0.000, E1   +36.054, E3 +241366.675}
SPL {X  -160.000, Y  +601.495, Z    +0.000, E1   +56.174, E3 +241387.604}
SPL {X  -160.000, Y  +515.545, Z    +0.000, E1   +60.629, E3 +241462.998}
SPL {X  -160.000, Y  +503.330, Z    +0.000, E1   +60.630, E3 +241477.604}
SPL {X  -160.000, Y  +487.139, Z    +0.000, E1   +60.676, E3 +241496.872}
SPL {X  -160.000, Y  +466.770, Z    +0.000, E1   +60.698, E3 +241521.167}
SPL {X  -160.000, Y  +454.269, Z    +0.000, E1   +59.898, E3 +241541.418}
ENDSPLINE

SPLINE
SPL {X  -160.000, Y  +458.973, Z    +0.000, E1   +55.880, E3 +241562.337}
ENDSPLINE

SPLINE
SPL {X  -160.000, Y  +435.816, Z    +0.000, E1   +57.237, E3 +241586.012}
SPL {X  -160.000, Y  +411.824, Z    +0.000, E1   +58.675, E3 +241608.506}
ENDSPLINE

SLIN {X  -200.000, Y  +533.000, E1    +0.000}
HALT
END
